FUNCTION_BLOCK FB_Light

VAR
	bColor1 AT %Q* : BYTE := 1;
	bColor2 AT %Q* : BYTE := 0;
	bFlashRate AT %Q* : BYTE := 1;
	bColor1Intensity AT %Q* : BYTE := 1;
	bColor2Intensity AT %Q* : BYTE := 1;
	bAudibleMode AT %Q* : BYTE := 0;
	bAnimationMode AT %Q* : BYTE := 1;
	bRotationalMode AT %Q* : BYTE := 0;

	tonTimerDelay1 : TON := (PT := T#500MS);
	tonTimerDelay2 : TON := (PT := T#500MS);
	
	nColorIndex : BYTE := 0;
END_VAR

METHOD mActivate : BOOL

VAR_INPUT
	inputVariable : BOOL;
END_VAR

VAR_INST
	localVar : BOOL;
END_VAR
localVar := inputVariable;

IF localVar THEN
	bAnimationMode := 1;
ELSE
	bAnimationMode := 0;
END_IF
END_METHOD

METHOD mCheckStatus : BOOL
VAR_INPUT
	bInputStatus : BOOL;
END_VAR



VAR
	tonTimeDelay : TON := (PT := T#4S);
END_VAR
IF bInputStatus THEN
	bColor1 := 0;
ELSE
	bColor1 := 1;
END_IF
END_METHOD

METHOD mFillArray : BOOL

VAR_INPUT
	//
END_VAR

VAR
	nIndex : INT := 1;
END_VAR

//FOR nIndex := 1 TO SIZEOF(aColors) DO
	//aColors[nIndex] := nIndex;
//END_FOR
END_METHOD

METHOD mLightDelay : BOOL

VAR_INPUT
	bInputState : BOOL; // case reset button from input
END_VAR

VAR_INST
	nCaseState : INT := 1;
	trigger : R_TRIG;
	
END_VAR
CASE nCaseState OF
	1:
		tonTimerDelay1(IN := TRUE);	
		IF tonTimerDelay1.Q THEN
			bColor1 := 1; // RED
			tonTimerDelay1(IN := FALSE);
			nCaseState := 2;
		END_IF

	2:
		tonTimerDelay2(IN := TRUE);
		IF tonTimerDelay2.Q THEN
			bColor1 := 0; // GREEN
			tonTimerDelay2(IN := FALSE);
			nCaseState := 1;
		END_IF
	
END_CASE
END_METHOD

METHOD mLightSpectrum : BOOL

VAR_INPUT
	//bInputState : BOOL; // case reset button from input
END_VAR

VAR_INST
	nCaseState : INT := 1;
	trigger : R_TRIG;
	
END_VAR
CASE nCaseState OF
	1:
		tonTimerDelay1(IN := TRUE);	
		IF tonTimerDelay1.Q THEN
			IF nColorIndex > 12 THEN
				nColorIndex := 0;
			END_IF
			bColor1 := nColorIndex;
			nColorIndex := nColorIndex + 1;
			
			tonTimerDelay1(IN := FALSE);
			nCaseState := 2;
		END_IF

	2:
		tonTimerDelay2(IN := TRUE);
		IF tonTimerDelay2.Q THEN
			IF nColorIndex > 12 THEN
				nColorIndex := 0;
			END_IF
			bColor1 := nColorIndex;
			nColorIndex := nColorIndex + 1;

			tonTimerDelay2(IN := FALSE);
			nCaseState := 1;
		END_IF
	
END_CASE
END_METHOD

METHOD mSetAnimation : BOOL

VAR_INPUT
	bInputValue : BYTE;
END_VAR
bAnimationMode := bInputValue;
END_METHOD

METHOD mSetColor : BOOL

VAR_INPUT
	nInputNumber : INT;
END_VAR

bColor1 := INT_TO_BYTE(nInputNumber);
END_METHOD

END_FUNCTION_BLOCK

(* stored: Version 1.1.0.1, ProductVersion 3.1.4024.12
   POU FB_Light: Id {3343f800-a989-4948-9ef8-705ba864a91b}, SpecialFunc None
   Method mActivate: Id {e5387f86-92eb-4bf1-b863-10dd15db2427}
   Method mCheckStatus: Id {839dd1cb-c416-4d9d-be4a-9570ed6c2e95}
   Method mFillArray: Id {7e5dd064-c880-4db2-bb4a-e034369fae43}
   Method mLightDelay: Id {79d56d5c-f543-437f-819f-536c881341e0}
   Method mLightSpectrum: Id {00b33b1f-8844-4e0a-b32f-528ac7697605}
   Method mSetAnimation: Id {01860b90-909a-43c9-9728-9496cf596de0}
   Method mSetColor: Id {d7d90027-3049-4483-8c5e-d6bc90596754} *)
